
// ===== library: MasterCopy "Homing_V90PN" =====

FUNCTION_BLOCK "Homing_V90PN"   // FB38001, SCL
{ S7_Optimized_Access := 'TRUE' }
VERSION : 0.1
   VAR_INPUT
      RefMode : Int;
      Off1 : Bool;
      AckError : Bool;
      Execute : Bool;
      RefDir : Bool;
      RefCam : Bool;
      HWLimitActive : Bool;
      RefCamPin : Int;
      HW_ID : Hw_Io;
   END_VAR
   VAR_OUTPUT
      Error : Bool;
      ErrorInfo : Word;
      RefOK : Bool;
   END_VAR
   VAR
      sxSendBuf : Struct
         STW1 : Word := 16#043e;
         EPosSTW1 : Word;
         EPosSTW2 : Word;
         STW2 : Word;
         OverrideV : Word := 16#4000;
         Position : DInt;
         Velocity : DInt;
         OverrideA : Word := 16#4000;
         OverrideD : Word := 16#4000;
         Reserve : Word;
      END_STRUCT;
      sxRecvBuf : Struct
         ZSW1 : Word;
         EPosZSW1 : Word;
         EPosZSW2 : Word;
         ZSW2 : Word;
         MELDW : Word;
         Position : DInt;
         Velocity : DInt;
         ErrNr : Word;
         WarnNr : Word;
         Reserve : Word;
      END_STRUCT;
      sbSignalFromDrive : Bool;
      swDiagID : Word;
      sbRefCam : Bool;
      sbRefDir : Bool;
      sbExecute : Bool := 1;
      sbExecuteFlag : Bool;
      sbExecuteRisingFlag : Bool;
      sbDriveEnabled : Bool;
      sbSetREF : Bool;
      sbOff1 : Bool := 1;
      sbAckError : Bool;
      sbCWLActive : Bool;
      sbCCWLActive : Bool;
      sbDriveFault : Bool;
      sbDriveReady : Bool;
      sbHWLimitActive : Bool := 1;
      sbJog1 : Bool;
      sbJog2 : Bool;
      sbModeFlag : Bool;
      sbRefCamRisingFlag : Bool;
      sbRefAction : Bool;
      sbRefCamFallingFlag : Bool;
      sbRefOk : Bool;
      sbJogToRef : Bool;
      sbJogEnabled : Bool;
      sbRefCamFalling : F_TRIG;
      sbRefCamRising : R_TRIG;
      sbExecuteRising : R_TRIG;
   END_VAR
   VAR_TEMP
      piRetSFC : Int;
      piCount : Int;
      swSendBuf : Array[0..11] of Word;
      swRecvBuf : Array[0..11] of Word;
   END_VAR
BEGIN
   // Author:   MC GMC MP ASIA
   // Version:  V1.0
   // Email:    mc_gmc_mp_asia.cn@siemens.com
   // Language: English only
   // 

   // Check the RefMode setting
   IF #RefMode < 0 OR #RefMode > 11 THEN
       #Error := true;
       #ErrorInfo := 16#8000;
   ELSE
       #Error := false;
       #ErrorInfo := 16#0000;
   END_IF;

   // Check which mode the signal is from drive

   IF #RefMode = 3 OR #RefMode = 5 OR #RefMode = 8 OR #RefMode = 10 THEN
       #sbSignalFromDrive := true;
   ELSE
       #sbSignalFromDrive := false;
   END_IF;

   // Check the RefCamPin seeting if needed
   IF #Error = false AND #sbSignalFromDrive=true  THEN
       IF #RefCamPin < 1 OR #RefCamPin > 4 THEN
           #Error := true;
           #ErrorInfo := 16#8010;
       ELSE
           #Error := false;
           #ErrorInfo := 16#0000;
       END_IF;
   END_IF;

   // Receive Signal from the drive
   #piRetSFC := DPRD_DAT(LADDR := #HW_ID, RECORD => #swRecvBuf);
   #swDiagID := INT_TO_WORD(#piRetSFC);

   //check the receiving communication error
   IF #piRetSFC<>0 AND #Error =false THEN
       #Error := true;
       #ErrorInfo := #swDiagID;
   ELSE
       #sxRecvBuf.Reserve := #swRecvBuf[11];
       #sxRecvBuf.EPosZSW1 := #swRecvBuf[1];
       #sxRecvBuf.ZSW1 := #swRecvBuf[0];
       #sbRefOk := #sxRecvBuf.ZSW1.%X11;
       #sbCWLActive := #sxRecvBuf.EPosZSW1.%X9;
       #sbCCWLActive := #sxRecvBuf.EPosZSW1.%X8;
       #sbDriveFault := #sxRecvBuf.ZSW1.%X3;
       #sbDriveReady := #sxRecvBuf.ZSW1.%X0;
       #sbDriveEnabled := #sxRecvBuf.ZSW1.%X2;
       #sbJogEnabled := #sxRecvBuf.EPosZSW1.%X10;


       // RefMode=0
       IF #RefMode = 0 THEN
           #sbRefCam := #RefCam;
           #sbRefDir := #RefDir;
           #sbHWLimitActive := #HWLimitActive;
           #sbSetREF := false;
           #sbExecuteFlag := FALSE;
           #sbExecute := true;

       // RefMode=1    
       ELSIF #RefMode=1 THEN
           #sbRefCam := FALSE;
           #sbRefDir := #RefDir;
           #sbHWLimitActive := #HWLimitActive;
           #sbSetREF := false;
           #sbExecuteFlag := FALSE;
           #sbExecute := true;

       //RefMode=2    
       ELSIF #RefMode=2 THEN
           #sbRefCam := FALSE;
           #sbRefDir := #RefDir;
           #sbHWLimitActive := #HWLimitActive;
           #sbSetREF := #Execute;
           #sbExecuteFlag := FALSE;
           #sbExecute := false;

       //RefMode=3    
       ELSIF #RefMode=3 THEN
           #sbRefDir := #RefDir;
           #sbHWLimitActive := #HWLimitActive;
           #sbSetREF := false;
           #sbExecuteFlag := FALSE;
           #sbExecute := true;

           IF #RefCamPin = 1 THEN
               #sbRefCam := #sxRecvBuf.Reserve.%X0;
           ELSIF #RefCamPin = 2 THEN
               #sbRefCam := #sxRecvBuf.Reserve.%X1;
           ELSIF #RefCamPin = 3 THEN
               #sbRefCam := #sxRecvBuf.Reserve.%X2;
           ELSIF #RefCamPin = 4 THEN
               #sbRefCam := #sxRecvBuf.Reserve.%X3;
           ELSE
               #sbRefCam := false;
           END_IF;

       //RefMode=4    
       ELSIF #RefMode=4 THEN
           #sbRefDir := #RefDir;
           #sbRefCam := #RefCam;
           #sbSetREF := false;
           #sbExecuteFlag := FALSE;
           #sbHWLimitActive := #HWLimitActive;

           IF #sbModeFlag = false THEN
               #sbExecute := true;
           END_IF;

           IF #sbCWLActive = true OR #sbCCWLActive = true THEN
               #sbExecute := false;
               #sbOff1 := false;
               #sbAckError := true;
               #sbModeFlag := true;
           END_IF;
           IF #sbModeFlag = true THEN
               IF #sbDriveFault = false AND #sbDriveReady = true THEN
                   #sbAckError := false;
                   #sbOff1 := true;
               END_IF;
               IF #sbCWLActive = true AND #sbDriveEnabled = true THEN
                   #sbJog1 := true;
                   #sbJog2 := false;
               END_IF;
               IF #sbCCWLActive = true AND #sbDriveEnabled = true THEN
                   #sbJog1 := false;
                   #sbJog2 := true;
               END_IF;

               #sbRefCamFalling(CLK := #sbRefCam,
                                         Q => #sbRefCamFallingFlag);

                   IF #sbJogToRef = true AND #sbJogEnabled=false THEN
                       #sbJogToRef := false;
                       #sbExecute := true;
                   END_IF;
               IF #sbRefCamFallingFlag = true THEN
                   #sbJog1 := false;
                   #sbJog2 := FALSE;
                   #sbJogToRef := true;
                   #sbRefCamFallingFlag := false;
               END_IF;
           END_IF;
           IF #sbRefOk = true OR #Execute = false THEN
               #sbModeFlag := false;
           END_IF;

       //RefMode=5    
       ELSIF #RefMode=5 THEN
           #sbExecuteFlag := FALSE;
           #sbSetREF := false;
           #sbRefDir := #RefDir;
           #sbHWLimitActive := #HWLimitActive;

           IF #sbModeFlag = false THEN
               #sbExecute := true;
           END_IF;

           IF #RefCamPin = 1 THEN
               #sbRefCam := #sxRecvBuf.Reserve.%X0;
           ELSIF #RefCamPin = 2 THEN
               #sbRefCam := #sxRecvBuf.Reserve.%X1;
           ELSIF #RefCamPin = 3 THEN
               #sbRefCam := #sxRecvBuf.Reserve.%X2;
           ELSIF #RefCamPin = 4 THEN
               #sbRefCam := #sxRecvBuf.Reserve.%X3;
           ELSE
               #sbRefCam := false;
           END_IF;

           IF #sbCWLActive = true OR #sbCCWLActive = true THEN
               #sbExecute := false;
               #sbOff1 := false;
               #sbAckError := true;
               #sbModeFlag := true;
           END_IF;
           IF #sbModeFlag = true THEN
               IF #sbDriveFault = false AND #sbDriveReady = true THEN
                   #sbAckError := false;
                   #sbOff1 := true;
               END_IF;
               IF #sbCWLActive = true AND #sbDriveEnabled = true THEN
                   #sbJog1 := true;
                   #sbJog2 := false;
               END_IF;
               IF #sbCCWLActive = true AND #sbDriveEnabled = true THEN
                   #sbJog1 := false;
                   #sbJog2 := true;
               END_IF;
               #sbRefCamFalling(CLK := #sbRefCam,
                                     Q => #sbRefCamFallingFlag);
               IF #sbJogToRef = true AND #sbJogEnabled = false THEN
                   #sbJogToRef := false;
                   #sbExecute := true;
               END_IF;
               IF #sbRefCamFallingFlag = true THEN
                   #sbJog1 := false;
                   #sbJog2 := FALSE;
                   #sbJogToRef := true;
                   #sbRefCamFallingFlag := false;
               END_IF;

           END_IF;
           IF #sbRefOk = true OR #Execute = false THEN
               #sbModeFlag := false;
           END_IF;

       //RefMode=6
       ELSIF #RefMode=6 THEN
           #sbRefDir := #RefDir;
           #sbSetREF := false;
           #sbExecuteFlag := FALSE;
           #sbExecute:=true;

           IF #RefCamPin = 1 THEN
               #sbRefCam := NOT #sxRecvBuf.Reserve.%X0;
           ELSIF #RefCamPin = 2 THEN
               #sbRefCam := NOT #sxRecvBuf.Reserve.%X1;
           ELSIF #RefCamPin = 3 THEN
               #sbRefCam := NOT #sxRecvBuf.Reserve.%X2;
           ELSIF #RefCamPin = 4 THEN
               #sbRefCam := NOT #sxRecvBuf.Reserve.%X3;
           ELSE
               #sbRefCam := false;
           END_IF;

           IF #HWLimitActive = true THEN
               IF #sbExecute = true AND #sbRefOk = false THEN
                   #sbHWLimitActive := FALSE;
               ELSE
                   #sbHWLimitActive := true;
               END_IF;
           END_IF;

       //RefMode=7    
       ELSIF #RefMode=7 THEN
           #sbRefDir := #RefDir;
           #sbRefCam := #RefCam;
           #sbExecute := FALSE;
           #sbRefCamRising(CLK := #sbRefCam,
                                Q => #sbRefCamRisingFlag);
           #sbExecuteRising(CLK := #Execute,
                                 Q => #sbExecuteRisingFlag);
           IF #sbExecuteRisingFlag = true THEN
               #sbExecuteFlag := true;
           END_IF;
           IF #sbExecuteFlag=true  AND #Execute= true THEN
               IF #sbRefDir = false THEN
                   #sbJog1 := FALSE;
                   #sbJog2 := true;
               ELSE
                   #sbJog1 := TRUE;
                   #sbJog2 := false;
               END_IF;
               IF #sbRefCamRisingFlag = true THEN
                   #sbJog1 := false;
                   #sbJog2 := false;
                   #sbSetREF := #sbExecuteFlag;
                   #sbRefAction := true;
               END_IF;
           ELSE
               #sbJog1 := false;
               #sbJog2 := false;
           END_IF;
           IF #sbExecuteFlag = true AND #sbRefOk = true AND #sbRefAction =true THEN
               #sbExecuteFlag := false;
               #sbRefAction := false;
           END_IF;
       //RefMode=8
       ELSIF #RefMode=8 THEN
           #sbRefDir := #RefDir;
           #sbExecute := FALSE;
           IF #RefCamPin = 1 THEN
               #sbRefCam := #sxRecvBuf.Reserve.%X0;
           ELSIF #RefCamPin = 2 THEN
               #sbRefCam := #sxRecvBuf.Reserve.%X1;
           ELSIF #RefCamPin = 3 THEN
               #sbRefCam := #sxRecvBuf.Reserve.%X2;
           ELSIF #RefCamPin = 4 THEN
               #sbRefCam := #sxRecvBuf.Reserve.%X3;
           ELSE
               #sbRefCam := false;
           END_IF;

           #sbRefCamRising(CLK := #sbRefCam,
                                Q => #sbRefCamRisingFlag);
           #sbExecuteRising(CLK := #Execute,
                                 Q => #sbExecuteRisingFlag);
           IF #sbExecuteRisingFlag = true THEN
               #sbExecuteFlag := true;
           END_IF;
           IF #sbExecuteFlag =true AND #Execute= true THEN
               IF #sbRefDir = false THEN
                   #sbJog1 := FALSE;
                   #sbJog2 := true;
               ELSE
                   #sbJog1 := TRUE;
                   #sbJog2 := false;
               END_IF;
               IF #sbRefCamRisingFlag = true THEN
                   #sbJog1 := false;
                   #sbJog2 := false;
                   #sbSetREF := #sbExecuteFlag;
                   #sbRefAction := true;
               END_IF;
           ELSE
               #sbJog1 := false;
               #sbJog2 := false;
           END_IF;
           IF #sbExecuteFlag = true AND #sbRefOk = true AND #sbRefAction = true THEN
               #sbExecuteFlag := false;
               #sbRefAction := false;
           END_IF;

       //RefMode=9
       ELSIF #RefMode=9 THEN
           #sbExecute := false;
           #sbRefCam := #RefCam;
           #sbRefDir := #RefDir;
           #sbHWLimitActive := #HWLimitActive;

           #sbRefCamRising(CLK := #sbRefCam,
                               Q => #sbRefCamRisingFlag);
           #sbExecuteRising(CLK := #Execute,
                                Q => #sbExecuteRisingFlag);
           IF #sbExecuteRisingFlag = true THEN
               #sbExecuteFlag := true;
           END_IF;
           IF #sbModeFlag = false THEN
               IF #sbExecuteFlag = true AND #Execute = true THEN
                   IF #sbRefDir = false THEN
                       #sbJog1 := FALSE;
                       #sbJog2 := true;
                   ELSE
                       #sbJog1 := TRUE;
                       #sbJog2 := false;
                   END_IF;
                   IF #sbRefCamRisingFlag = true THEN
                       #sbJog1 := false;
                       #sbJog2 := false;
                       #sbSetREF := #sbExecuteFlag;
                       #sbRefAction := true;
                   END_IF;
               ELSE
                   #sbJog1 := false;
                   #sbJog2 := false;
               END_IF;
           END_IF;
           IF #sbExecuteFlag = true AND #sbRefOk = true AND #sbRefAction = true THEN
               #sbExecuteFlag := false;
               #sbRefAction := false;
           END_IF;

           IF #sbCWLActive = true OR #sbCCWLActive = true THEN
               #sbExecuteFlag := false;
               #sbOff1 := false;
               #sbAckError := true;
               #sbModeFlag := true;
           END_IF;
           IF #sbModeFlag = true THEN
               IF #sbDriveFault = false AND #sbDriveReady = true THEN
                   #sbAckError := false;
                   #sbOff1 := true;
               END_IF;
               IF #sbCWLActive = true AND #sbDriveEnabled = true THEN
                   #sbJog1 := true;
                   #sbJog2 := false;
               END_IF;
               IF #sbCCWLActive = true AND #sbDriveEnabled = true THEN
                   #sbJog1 := false;
                   #sbJog2 := true;
               END_IF;

               #sbRefCamFalling(CLK := #sbRefCam,
                                     Q => #sbRefCamFallingFlag);

               IF #sbJogToRef = true AND #sbJogEnabled = false THEN
                   #sbJogToRef := false;
                   #sbExecuteFlag := true;
                   #sbModeFlag := false;
               END_IF;
               IF #sbRefCamFallingFlag = true THEN
                   #sbJog1 := false;
                   #sbJog2 := FALSE;
                   #sbJogToRef := true;
                   #sbRefCamFallingFlag := false;
               END_IF;
           END_IF;

       //RefMode=10
       ELSIF #RefMode=10 THEN
           #sbExecute := false;
           #sbHWLimitActive := #HWLimitActive;
           #sbRefDir := #RefDir;
           IF #RefCamPin = 1 THEN
               #sbRefCam :=  #sxRecvBuf.Reserve.%X0;
           ELSIF #RefCamPin = 2 THEN
               #sbRefCam :=  #sxRecvBuf.Reserve.%X1;
           ELSIF #RefCamPin = 3 THEN
               #sbRefCam :=  #sxRecvBuf.Reserve.%X2;
           ELSIF #RefCamPin = 4 THEN
               #sbRefCam :=  #sxRecvBuf.Reserve.%X3;
           ELSE
               #sbRefCam := false;
           END_IF;
           #sbHWLimitActive := #HWLimitActive;

           #sbRefCamRising(CLK := #sbRefCam,
                               Q => #sbRefCamRisingFlag);
           #sbExecuteRising(CLK := #Execute,
                                Q => #sbExecuteRisingFlag);
           IF #sbExecuteRisingFlag = true THEN
               #sbExecuteFlag := true;
           END_IF;
           IF #sbModeFlag = false THEN
               IF #sbExecuteFlag = true AND #Execute = true THEN
                   IF #sbRefDir = false THEN
                       #sbJog1 := FALSE;
                       #sbJog2 := true;
                   ELSE
                       #sbJog1 := TRUE;
                       #sbJog2 := false;
                   END_IF;
                   IF #sbRefCamRisingFlag = true THEN
                       #sbJog1 := false;
                       #sbJog2 := false;
                       #sbSetREF := #sbExecuteFlag;
                       #sbRefAction := true;
                   END_IF;
               ELSE
                   #sbJog1 := false;
                   #sbJog2 := false;
               END_IF;
           END_IF;
           IF #sbExecuteFlag = true AND #sbRefOk = true AND #sbRefAction = true THEN
               #sbExecuteFlag := false;
               #sbRefAction := false;
           END_IF;

           IF #sbCWLActive = true OR #sbCCWLActive = true THEN
               #sbExecuteFlag := false;
               #sbOff1 := false;
               #sbAckError := true;
               #sbModeFlag := true;
           END_IF;
           IF #sbModeFlag = true THEN
               IF #sbDriveFault = false AND #sbDriveReady = true THEN
                   #sbAckError := false;
                   #sbOff1 := true;
               END_IF;
               IF #sbCWLActive = true AND #sbDriveEnabled = true THEN
                   #sbJog1 := true;
                   #sbJog2 := false;
               END_IF;
               IF #sbCCWLActive = true AND #sbDriveEnabled = true THEN
                   #sbJog1 := false;
                   #sbJog2 := true;
               END_IF;

               #sbRefCamFalling(CLK := #sbRefCam,
                                    Q => #sbRefCamFallingFlag);

               IF #sbJogToRef = true AND #sbJogEnabled = false THEN
                   #sbJogToRef := false;
                   #sbExecuteFlag := true;
                   #sbModeFlag := false;
               END_IF;
               IF #sbRefCamFallingFlag = true THEN
                   #sbJog1 := false;
                   #sbJog2 := FALSE;
                   #sbJogToRef := true;
                   #sbRefCamFallingFlag := false;
               END_IF;
           END_IF;

       // RefMode is not existed.
       ELSE
           #sbExecute := false ;
           #sbRefCam := FALSE;
           #sbRefDir := FALSE;
           #sbAckError := false;
           #sbOff1 := FALSE;
           #sbHWLimitActive := FALSE;
           #sbSetREF := false;
           #sbExecuteFlag := FALSE;
       END_IF;

   END_IF;

   //Send data
   #sxSendBuf.STW1.%X0 := #sbOff1 AND #Off1;
   #sxSendBuf.STW1.%X7 := #sbAckError OR #sbAckError;
   #sxSendBuf.STW1.%X8 := #sbJog1;
   #sxSendBuf.STW1.%X9 := #sbJog2;
   #sxSendBuf.STW1.%X11 := #sbExecute AND #Execute;
   #sxSendBuf.EPosSTW2.%X1 := #sbSetREF;
   #sxSendBuf.EPosSTW2.%X2 := #sbRefCam;
   #sxSendBuf.EPosSTW2.%X9 := #sbRefDir;
   #sxSendBuf.EPosSTW2.%X15 := #sbHWLimitActive AND #HWLimitActive;

   #swSendBuf[0] := #sxSendBuf.STW1;
   #swSendBuf[1] := #sxSendBuf.EPosSTW1;
   #swSendBuf[2] := #sxSendBuf.EPosSTW2;
   #swSendBuf[3] := #sxSendBuf.STW2;
   #swSendBuf[4] := #sxSendBuf.OverrideV;
   #swSendBuf[5] := #sxSendBuf.Position.%W1;
   #swSendBuf[6] := #sxSendBuf.Position.%W0;
   #swSendBuf[7] := #sxSendBuf.Velocity.%W1;
   #swSendBuf[8] := #sxSendBuf.Velocity.%W0;
   #swSendBuf[9] := #sxSendBuf.OverrideA;
   #swSendBuf[10] := #sxSendBuf.OverrideD;
   #swSendBuf[11] := #sxSendBuf.Reserve;

   //send the command to the drive
   IF #Error = false THEN
       #piRetSFC := DPWR_DAT(LADDR := #HW_ID, RECORD := #swSendBuf);
       #swDiagID := INT_TO_WORD(#piRetSFC);
   END_IF;

   IF #piRetSFC <> 0 AND #Error = false THEN
       #Error := true;
       #ErrorInfo := #swDiagID;
   END_IF;

   #RefOK := #sbRefOk;
END_FUNCTION_BLOCK